// TIA Portal V18 export
TYPE "UDT_TrackingReport_HMI_OP1"
// stored: IsFailsafeCompliant false
   STRUCT
      ClearReport : Bool;   // 清除数据命令
      PosInx_HMI : Int;   // 触摸屏页面位置
      PageNo : Int;   // 触摸屏页面编号
      RowIndex : Array[0..9] of Int;   // 行号
      TrackingReport : Array[0..9] of "UDT_TrackingReport_OP01";   // HMI显示数据
   END_STRUCT;
END_TYPE
